// TwinCAT 3 PLC project M1L1_PLC
// ProgramVersion: 3.1.4022.7
// libraries:
//   LCLS General, * (SLAC)
//   Tc2_ControllerToolbox, * (Beckhoff Automation GmbH)
//   Tc2_MC2, * (Beckhoff Automation GmbH)
//   Tc2_SerialCom, * (Beckhoff Automation GmbH)
//   Tc2_Standard, * (Beckhoff Automation GmbH)
//   Tc2_System, * (Beckhoff Automation GmbH)
//   Tc2_Utilities, * (Beckhoff Automation GmbH)
//   Tc3_Module, * (Beckhoff Automation GmbH)
//   VisuDialogs
//   lcls-twincat-motion,0.0.0,SLAC
// project tree:
//   Common/DUTs/ E_PiezoControl.TcDUT (not stored), E_PitchControl.TcDUT (not stored), HOMS_PitchMechanism.TcDUT, ST_AbstractAxis.TcDUT (not stored), ST_HOMSStepper.TcDUT (not stored), ST_PiezoAxis.TcDUT
//   Common/POUs/Helpers/ FB_PI_E621_SerialDriver.TcPOU (not stored), FB_PI_E621_SerialTransaction.TcPOU (not stored), MC_SmoothMover.TcPOU (not stored), WithinRange.TcPOU (not stored)
//   Common/POUs/HOMS_FBs/ FB_PiezoControl.TcPOU (not stored), FB_PitchControl.TcPOU (not stored)
//   DUTs/ DUT_MotionStage_Extras.TcDUT (not stored)
//   / GlobalTextList.TcGTLO, PiezoDriver.TcTTO, PlcTask.TcTTO (not stored), Visualization Manager.TcVMO (not stored)
//   GVLs/ GVL_COM_Buffers.TcGVL (not stored), GVL_Constants.TcGVL (not stored), GVL_Devices.TcGVL, GVL_SerialIO.TcGVL (not stored)
//   POUs/ MAIN.TcPOU
//   POUs/Serial Comm/ PiezoSerial.TcPOU (not stored), P_Serial_Com.TcPOU (not stored)
//   VISUs/ Visualization.TcVIS, VISU_MotionStage.TcVIS
// real-time tasks:
//   TASK PlcTask: cycle T#10ms, priority 20, ADS port 350
//   TASK serial_com: cycle T#10ms, priority 21, ADS port 351
//   TASK PiezoDriver: cycle T#1ms, priority 3, ADS port 352
//   TASK SerialIO: cycle T#2ms, priority 1, ADS port 353
// motion (NC):
//   TASK NC-Task 1 SAF: cycle T#2ms, priority 4, ADS port 501
//   TASK NC-Task 1 SVB: cycle T#10ms, priority 8, ADS port 511
//   AXIS y_up (id 6)
//     General: UnitName=um
//     Dynamic: Acceleration=5050, Deceleration=5050, Jerk=5100500, DelayTime=0.008
//     Velo: Maximum=100
//     OtherSettings: AllowMotionCmdToSlave=true
//     encoder EncType=29
//       EncPara: ScaleFactorNumerator=1, ScaleFactorDenominator=1000, MaxCount=#xffffffff
//         SoftEndMinControl: Enable=true, Range=10000
//         SoftEndMaxControl: Enable=true, Range=79999
//         Inc: RefSoftSyncMask=#x0000ffff
//     drive DrvType=24
//       DrvPara: Inverse=true
//         Analog: VeloReferenz=500
//         TimeComp: TaskDelayCycles=1
//     controller CtrType=3
//       CtrPara: PriorControlFactor=1
//         PosDiffControl: Range=50, Time=0.2
//         PID: PosTn=0.005, PosIOutputLimit=0.0001, PosDOutputLimit=0, PosIDisableWhenMoving=true, DeadBandPosition=0.001
//         Observer: BandWidth=20
//   AXIS y_dwn (id 7)
//     General: UnitName=um
//     Dynamic: Acceleration=5050, Deceleration=5050, Jerk=5100500, DelayTime=0.008
//     Velo: Maximum=100
//     OtherSettings: AllowMotionCmdToSlave=true
//     encoder EncType=29
//       EncPara: ScaleFactorNumerator=1, ScaleFactorDenominator=1000, MaxCount=#xffffffff
//         SoftEndMinControl: Enable=true, Range=9000
//         SoftEndMaxControl: Enable=true, Range=79551
//         Inc: RefSoftSyncMask=#x0000ffff
//     drive DrvType=24
//       DrvPara: Inverse=true
//         Analog: VeloReferenz=500
//         TimeComp: TaskDelayCycles=1
//     controller CtrType=3
//       CtrPara: PriorControlFactor=1
//         PosDiffControl: Range=50, Time=0.2
//         PID: PosTn=0.005, PosIOutputLimit=0.0001, PosDOutputLimit=0, PosIDisableWhenMoving=true, DeadBandPosition=0.001
//         Observer: BandWidth=20
//   AXIS x_up (id 8)
//     General: UnitName=um
//     Dynamic: AccelerationMaximum=1000, DecelerationMaximum=1000, Acceleration=1000, Deceleration=1000, Jerk=5000, DelayTime=0.008
//     Velo: Maximum=300
//     OtherSettings: AllowMotionCmdToSlave=true
//     encoder EncType=29
//       EncPara: ScaleFactorNumerator=1, ScaleFactorDenominator=1000, MaxCount=#xffffffff
//         SoftEndMinControl: Enable=true, Range=16300
//         SoftEndMaxControl: Enable=true, Range=23200
//         Inc: RefSoftSyncMask=#x0000ffff
//     drive DrvType=24
//       DrvPara: Inverse=true
//         Analog: VeloReferenz=625
//         TimeComp: TaskDelayCycles=1
//     controller CtrType=3
//       CtrPara: PriorControlFactor=1
//         PosDiffControl: Range=50, Time=0.2
//         PID: PosTn=0.005, PosIOutputLimit=0.0001, PosDOutputLimit=0, PosIDisableWhenMoving=true, DeadBandPosition=0.001
//         Observer: BandWidth=20
//   AXIS x_dwn (id 9)
//     General: UnitName=um
//     Dynamic: AccelerationMaximum=1000, DecelerationMaximum=1000, Acceleration=1000, Deceleration=1000, Jerk=5000, DelayTime=0.008
//     Velo: Maximum=300
//     OtherSettings: AllowMotionCmdToSlave=true
//     encoder EncType=29
//       EncPara: ScaleFactorNumerator=1, ScaleFactorDenominator=1000, MaxCount=#xffffffff
//         SoftEndMinControl: Enable=true, Range=17400
//         SoftEndMaxControl: Enable=true, Range=24500
//         Inc: RefSoftSyncMask=#x0000ffff
//     drive DrvType=24
//       Analog: VeloReferenz=625
//       TimeComp: TaskDelayCycles=1
//     controller CtrType=3
//       CtrPara: PriorControlFactor=1
//         PosDiffControl: Range=50, Time=0.2
//         PID: PosTn=0.005, PosIOutputLimit=0.0001, PosDOutputLimit=0, PosIDisableWhenMoving=true, DeadBandPosition=0.001
//         Observer: BandWidth=20
//   AXIS pitch (id 10)
//     General: UnitName=urad
//     Dynamic: Acceleration=64082.2, Deceleration=64082.2, Jerk=711156, DelayTime=0.008
//     Velo: Maximum=50
//     OtherSettings: AllowMotionCmdToSlave=true
//     encoder EncType=29
//       EncPara: ScaleFactorNumerator=0.00556, MaxCount=#xffffffff
//         ActPosCorrection: Time=0.008
//         Inc: RefSoftSyncMask=#x0000ffff
//     drive DrvType=24
//       DrvPara: Inverse=true
//         Analog: VeloReferenz=7042.25
//         TimeComp: TaskDelayCycles=1
//     controller CtrType=3
//       CtrPara: PriorControlFactor=1
//         PosDiffControl: Range=15, Time=0.2
//         PID: PosKp=9, PosTn=0.0006, PosTv=1.2e-05, PosIOutputLimit=0.0005, PosDOutputLimit=0.0035, AccKa=0.001, DeadBandPosition=0.1
//         Observer: BandWidth=20
// I/O:
//   DEVICE Device 1 (EtherCAT)
//   DEVICE Device 4 (EtherCAT)
// variable links:
//   Axes/pitch <-> Device 4 (EtherCAT)/Term 4 (EK1100)/Term 10 (EL7047) - PitchCoarse
//     Drive/Inputs/In/nState1 @bit 3 <-> STM Status/Status/Error
//     Drive/Inputs/In/nState1 @bit 7 <-> STM Status/Status/Motor stall
//     Drive/Inputs/In/nState1 @bit 5 <-> STM Status/Status/Moving negative
//     Drive/Inputs/In/nState1 @bit 4 <-> STM Status/Status/Moving positive
//     Drive/Inputs/In/nState1 @bit 1 <-> STM Status/Status/Ready
//     Drive/Inputs/In/nState1 <-> STM Status/Status/Ready to enable
//     Drive/Inputs/In/nState1 @bit 6 <-> STM Status/Status/Torque reduced
//     Drive/Inputs/In/nState1 @bit 2 <-> STM Status/Status/Warning
//     Drive/Inputs/In/nState2 @bit 3 <-> STM Status/Status/Digital input 1
//     Drive/Inputs/In/nState2 @bit 4 <-> STM Status/Status/Digital input 2
//     Drive/Inputs/In/nState2 @bit 5 <-> STM Status/Status/Sync error
//     Drive/Inputs/In/nState2 @bit 7 <-> STM Status/Status/TxPDO Toggle
//     Drive/Inputs/In/nState4 @bit 1 <-> WcState/InputToggle
//     Drive/Inputs/In/nState4 <-> WcState/WcState
//     Drive/Outputs/Out/nCtrl1 <-> STM Control/Control/Enable
//     Drive/Outputs/Out/nCtrl1 @bit 2 <-> STM Control/Control/Reduce torque
//     Drive/Outputs/Out/nCtrl1 @bit 1 <-> STM Control/Control/Reset
//     Drive/Outputs/Out/nCtrl2 @bit 3 <-> STM Control/Control/Digital output 1
//     Drive/Outputs/Out/nDataOut2[0] <-> STM Velocity/Velocity
//   Axes/pitch <-> Device 4 (EtherCAT)/Term 4 (EK1100)/Term 13 (EL5042) - Pitch
//     Enc/Inputs/In/nComState @bit 1 <-> WcState/InputToggle
//     Enc/Inputs/In/nComState <-> WcState/WcState
//     Enc/Inputs/In/nDataIn1 <-> FB Inputs Channel 1/Position
//     Enc/Inputs/In/nState1 @bit 12 <-> FB Inputs Channel 1/Status/Diag
//     Enc/Inputs/In/nState1 @bit 1 <-> FB Inputs Channel 1/Status/Error
//     Enc/Inputs/In/nState1 @bit 14 <-> FB Inputs Channel 1/Status/Input cycle counter
//     Enc/Inputs/In/nState1 @bit 2 <-> FB Inputs Channel 1/Status/Ready
//     Enc/Inputs/In/nState1 @bit 13 <-> FB Inputs Channel 1/Status/TxPDO State
//     Enc/Inputs/In/nState1 <-> FB Inputs Channel 1/Status/Warning
//   Axes/x_dwn <-> Device 4 (EtherCAT)/Term 4 (EK1100)/Term 12 (EL5042) - X
//     Enc/Inputs/In/nComState @bit 1 <-> WcState/InputToggle
//     Enc/Inputs/In/nComState <-> WcState/WcState
//     Enc/Inputs/In/nDataIn1 <-> FB Inputs Channel 2/Position
//     Enc/Inputs/In/nState1 @bit 12 <-> FB Inputs Channel 2/Status/Diag
//     Enc/Inputs/In/nState1 @bit 1 <-> FB Inputs Channel 2/Status/Error
//     Enc/Inputs/In/nState1 @bit 14 <-> FB Inputs Channel 2/Status/Input cycle counter
//     Enc/Inputs/In/nState1 @bit 2 <-> FB Inputs Channel 2/Status/Ready
//     Enc/Inputs/In/nState1 @bit 13 <-> FB Inputs Channel 2/Status/TxPDO State
//     Enc/Inputs/In/nState1 <-> FB Inputs Channel 2/Status/Warning
//   Axes/x_dwn <-> Device 4 (EtherCAT)/Term 4 (EK1100)/Term 9 (EL7047) - Xdwn
//     Drive/Inputs/In/nState1 @bit 3 <-> STM Status/Status/Error
//     Drive/Inputs/In/nState1 @bit 7 <-> STM Status/Status/Motor stall
//     Drive/Inputs/In/nState1 @bit 5 <-> STM Status/Status/Moving negative
//     Drive/Inputs/In/nState1 @bit 4 <-> STM Status/Status/Moving positive
//     Drive/Inputs/In/nState1 @bit 1 <-> STM Status/Status/Ready
//     Drive/Inputs/In/nState1 <-> STM Status/Status/Ready to enable
//     Drive/Inputs/In/nState1 @bit 6 <-> STM Status/Status/Torque reduced
//     Drive/Inputs/In/nState1 @bit 2 <-> STM Status/Status/Warning
//     Drive/Inputs/In/nState2 @bit 3 <-> STM Status/Status/Digital input 1
//     Drive/Inputs/In/nState2 @bit 4 <-> STM Status/Status/Digital input 2
//     Drive/Inputs/In/nState2 @bit 5 <-> STM Status/Status/Sync error
//     Drive/Inputs/In/nState2 @bit 7 <-> STM Status/Status/TxPDO Toggle
//     Drive/Inputs/In/nState4 @bit 1 <-> WcState/InputToggle
//     Drive/Inputs/In/nState4 <-> WcState/WcState
//     Drive/Outputs/Out/nCtrl1 <-> STM Control/Control/Enable
//     Drive/Outputs/Out/nCtrl1 @bit 2 <-> STM Control/Control/Reduce torque
//     Drive/Outputs/Out/nCtrl1 @bit 1 <-> STM Control/Control/Reset
//     Drive/Outputs/Out/nCtrl2 @bit 3 <-> STM Control/Control/Digital output 1
//     Drive/Outputs/Out/nDataOut2[0] <-> STM Velocity/Velocity
//   Axes/x_up <-> Device 4 (EtherCAT)/Term 4 (EK1100)/Term 12 (EL5042) - X
//     Enc/Inputs/In/nComState @bit 1 <-> WcState/InputToggle
//     Enc/Inputs/In/nComState <-> WcState/WcState
//     Enc/Inputs/In/nDataIn1 <-> FB Inputs Channel 1/Position
//     Enc/Inputs/In/nState1 @bit 12 <-> FB Inputs Channel 1/Status/Diag
//     Enc/Inputs/In/nState1 @bit 1 <-> FB Inputs Channel 1/Status/Error
//     Enc/Inputs/In/nState1 @bit 14 <-> FB Inputs Channel 1/Status/Input cycle counter
//     Enc/Inputs/In/nState1 @bit 2 <-> FB Inputs Channel 1/Status/Ready
//     Enc/Inputs/In/nState1 @bit 13 <-> FB Inputs Channel 1/Status/TxPDO State
//     Enc/Inputs/In/nState1 <-> FB Inputs Channel 1/Status/Warning
//   Axes/x_up <-> Device 4 (EtherCAT)/Term 4 (EK1100)/Term 8 (EL7047) - Xup
//     Drive/Inputs/In/nState1 @bit 3 <-> STM Status/Status/Error
//     Drive/Inputs/In/nState1 @bit 7 <-> STM Status/Status/Motor stall
//     Drive/Inputs/In/nState1 @bit 5 <-> STM Status/Status/Moving negative
//     Drive/Inputs/In/nState1 @bit 4 <-> STM Status/Status/Moving positive
//     Drive/Inputs/In/nState1 @bit 1 <-> STM Status/Status/Ready
//     Drive/Inputs/In/nState1 <-> STM Status/Status/Ready to enable
//     Drive/Inputs/In/nState1 @bit 6 <-> STM Status/Status/Torque reduced
//     Drive/Inputs/In/nState1 @bit 2 <-> STM Status/Status/Warning
//     Drive/Inputs/In/nState2 @bit 3 <-> STM Status/Status/Digital input 1
//     Drive/Inputs/In/nState2 @bit 4 <-> STM Status/Status/Digital input 2
//     Drive/Inputs/In/nState2 @bit 5 <-> STM Status/Status/Sync error
//     Drive/Inputs/In/nState2 @bit 7 <-> STM Status/Status/TxPDO Toggle
//     Drive/Inputs/In/nState4 @bit 1 <-> WcState/InputToggle
//     Drive/Inputs/In/nState4 <-> WcState/WcState
//     Drive/Outputs/Out/nCtrl1 <-> STM Control/Control/Enable
//     Drive/Outputs/Out/nCtrl1 @bit 2 <-> STM Control/Control/Reduce torque
//     Drive/Outputs/Out/nCtrl1 @bit 1 <-> STM Control/Control/Reset
//     Drive/Outputs/Out/nCtrl2 @bit 3 <-> STM Control/Control/Digital output 1
//     Drive/Outputs/Out/nDataOut2[0] <-> STM Velocity/Velocity
//   Axes/y_dwn <-> Device 4 (EtherCAT)/Term 4 (EK1100)/Term 11 (EL5042) - Y
//     Enc/Inputs/In/nComState @bit 1 <-> WcState/InputToggle
//     Enc/Inputs/In/nComState <-> WcState/WcState
//     Enc/Inputs/In/nDataIn1 <-> FB Inputs Channel 2/Position
//     Enc/Inputs/In/nState1 @bit 12 <-> FB Inputs Channel 2/Status/Diag
//     Enc/Inputs/In/nState1 @bit 1 <-> FB Inputs Channel 2/Status/Error
//     Enc/Inputs/In/nState1 @bit 14 <-> FB Inputs Channel 2/Status/Input cycle counter
//     Enc/Inputs/In/nState1 @bit 2 <-> FB Inputs Channel 2/Status/Ready
//     Enc/Inputs/In/nState1 @bit 13 <-> FB Inputs Channel 2/Status/TxPDO State
//     Enc/Inputs/In/nState1 <-> FB Inputs Channel 2/Status/Warning
//   Axes/y_dwn <-> Device 4 (EtherCAT)/Term 4 (EK1100)/Term 7 (EL7047) - Ydwn
//     Drive/Inputs/In/nState1 @bit 3 <-> STM Status/Status/Error
//     Drive/Inputs/In/nState1 @bit 7 <-> STM Status/Status/Motor stall
//     Drive/Inputs/In/nState1 @bit 5 <-> STM Status/Status/Moving negative
//     Drive/Inputs/In/nState1 @bit 4 <-> STM Status/Status/Moving positive
//     Drive/Inputs/In/nState1 @bit 1 <-> STM Status/Status/Ready
//     Drive/Inputs/In/nState1 <-> STM Status/Status/Ready to enable
//     Drive/Inputs/In/nState1 @bit 6 <-> STM Status/Status/Torque reduced
//     Drive/Inputs/In/nState1 @bit 2 <-> STM Status/Status/Warning
//     Drive/Inputs/In/nState2 @bit 3 <-> STM Status/Status/Digital input 1
//     Drive/Inputs/In/nState2 @bit 4 <-> STM Status/Status/Digital input 2
//     Drive/Inputs/In/nState2 @bit 5 <-> STM Status/Status/Sync error
//     Drive/Inputs/In/nState2 @bit 7 <-> STM Status/Status/TxPDO Toggle
//     Drive/Inputs/In/nState4 @bit 1 <-> WcState/InputToggle
//     Drive/Inputs/In/nState4 <-> WcState/WcState
//     Drive/Outputs/Out/nCtrl1 <-> STM Control/Control/Enable
//     Drive/Outputs/Out/nCtrl1 @bit 2 <-> STM Control/Control/Reduce torque
//     Drive/Outputs/Out/nCtrl1 @bit 1 <-> STM Control/Control/Reset
//     Drive/Outputs/Out/nCtrl2 @bit 3 <-> STM Control/Control/Digital output 1
//     Drive/Outputs/Out/nDataOut2[0] <-> STM Velocity/Velocity
//   Axes/y_up <-> Device 4 (EtherCAT)/Term 4 (EK1100)/Term 11 (EL5042) - Y
//     Enc/Inputs/In/nComState @bit 1 <-> WcState/InputToggle
//     Enc/Inputs/In/nComState <-> WcState/WcState
//     Enc/Inputs/In/nDataIn1 <-> FB Inputs Channel 1/Position
//     Enc/Inputs/In/nState1 @bit 12 <-> FB Inputs Channel 1/Status/Diag
//     Enc/Inputs/In/nState1 @bit 1 <-> FB Inputs Channel 1/Status/Error
//     Enc/Inputs/In/nState1 @bit 14 <-> FB Inputs Channel 1/Status/Input cycle counter
//     Enc/Inputs/In/nState1 @bit 2 <-> FB Inputs Channel 1/Status/Ready
//     Enc/Inputs/In/nState1 @bit 13 <-> FB Inputs Channel 1/Status/TxPDO State
//     Enc/Inputs/In/nState1 <-> FB Inputs Channel 1/Status/Warning
//   Axes/y_up <-> Device 4 (EtherCAT)/Term 4 (EK1100)/Term 6 (EL7047) - Yup
//     Drive/Inputs/In/nState1 @bit 3 <-> STM Status/Status/Error
//     Drive/Inputs/In/nState1 @bit 7 <-> STM Status/Status/Motor stall
//     Drive/Inputs/In/nState1 @bit 5 <-> STM Status/Status/Moving negative
//     Drive/Inputs/In/nState1 @bit 4 <-> STM Status/Status/Moving positive
//     Drive/Inputs/In/nState1 @bit 1 <-> STM Status/Status/Ready
//     Drive/Inputs/In/nState1 <-> STM Status/Status/Ready to enable
//     Drive/Inputs/In/nState1 @bit 6 <-> STM Status/Status/Torque reduced
//     Drive/Inputs/In/nState1 @bit 2 <-> STM Status/Status/Warning
//     Drive/Inputs/In/nState2 @bit 3 <-> STM Status/Status/Digital input 1
//     Drive/Inputs/In/nState2 @bit 4 <-> STM Status/Status/Digital input 2
//     Drive/Inputs/In/nState2 @bit 5 <-> STM Status/Status/Sync error
//     Drive/Inputs/In/nState2 @bit 7 <-> STM Status/Status/TxPDO Toggle
//     Drive/Inputs/In/nState4 @bit 1 <-> WcState/InputToggle
//     Drive/Inputs/In/nState4 <-> WcState/WcState
//     Drive/Outputs/Out/nCtrl1 <-> STM Control/Control/Enable
//     Drive/Outputs/Out/nCtrl1 @bit 2 <-> STM Control/Control/Reduce torque
//     Drive/Outputs/Out/nCtrl1 @bit 1 <-> STM Control/Control/Reset
//     Drive/Outputs/Out/nCtrl2 @bit 3 <-> STM Control/Control/Digital output 1
//     Drive/Outputs/Out/nDataOut2[0] <-> STM Velocity/Velocity
//   M1L1_PLC Instance <-> Device 1 (EtherCAT)/Term 1 (EK1200)/Term 2 (EL1004)
//     PlcTask Inputs/MAIN.bSTOEnable1 <-> Channel 1/Input
//     PlcTask Inputs/MAIN.bSTOEnable2 <-> Channel 2/Input
//   M1L1_PLC Instance <-> Device 4 (EtherCAT)/Term 4 (EK1100)/Term 10 (EL7047) - PitchCoarse
//     PlcTask Inputs/GVL_Devices.M5.bLimitBackwardEnable <-> STM Status/Status/Digital input 2
//     PlcTask Inputs/GVL_Devices.M5.bLimitForwardEnable <-> STM Status/Status/Digital input 1
//   M1L1_PLC Instance <-> Device 4 (EtherCAT)/Term 4 (EK1100)/Term 11 (EL5042) - Y
//     PlcTask Inputs/MAIN.y_dwn_enc/Count <-> FB Inputs Channel 2/Position
//     PlcTask Inputs/MAIN.y_up_enc/Count <-> FB Inputs Channel 1/Position
//   M1L1_PLC Instance <-> Device 4 (EtherCAT)/Term 4 (EK1100)/Term 12 (EL5042) - X
//     PlcTask Inputs/MAIN.x_dwn_enc/Count <-> FB Inputs Channel 2/Position
//     PlcTask Inputs/MAIN.x_up_enc/Count <-> FB Inputs Channel 1/Position
//   M1L1_PLC Instance <-> Device 4 (EtherCAT)/Term 4 (EK1100)/Term 13 (EL5042) - Pitch
//     PlcTask Inputs/GVL_Devices.M1L0_Pitch.diEncCnt <-> FB Inputs Channel 1/Position
//   M1L1_PLC Instance <-> Device 4 (EtherCAT)/Term 4 (EK1100)/Term 14 (EL6001) - PitchFine
//     PlcTask Inputs/GVL_SerialIO.Serial_P1_stComIn/D[{0..21}] <-> COM Inputs/Data In {0..21}  (22 links)
//     PlcTask Inputs/GVL_SerialIO.Serial_P1_stComIn/Status <-> COM Inputs/Status
//     PlcTask Outputs/GVL_SerialIO.Serial_P1_stComOut/Ctrl <-> COM Outputs/Ctrl
//     PlcTask Outputs/GVL_SerialIO.Serial_P1_stComOut/D[{0..21}] <-> COM Outputs/Data Out {0..21}  (22 links)
//   M1L1_PLC Instance <-> Device 4 (EtherCAT)/Term 4 (EK1100)/Term 6 (EL7047) - Yup
//     PlcTask Inputs/GVL_Devices.M1.bLimitBackwardEnable <-> STM Status/Status/Digital input 2
//     PlcTask Inputs/GVL_Devices.M1.bLimitForwardEnable <-> STM Status/Status/Digital input 1
//   M1L1_PLC Instance <-> Device 4 (EtherCAT)/Term 4 (EK1100)/Term 7 (EL7047) - Ydwn
//     PlcTask Inputs/GVL_Devices.M2.bLimitBackwardEnable <-> STM Status/Status/Digital input 2
//     PlcTask Inputs/GVL_Devices.M2.bLimitForwardEnable <-> STM Status/Status/Digital input 1
//   M1L1_PLC Instance <-> Device 4 (EtherCAT)/Term 4 (EK1100)/Term 8 (EL7047) - Xup
//     PlcTask Inputs/GVL_Devices.M3.bLimitBackwardEnable <-> STM Status/Status/Digital input 2
//     PlcTask Inputs/GVL_Devices.M3.bLimitForwardEnable <-> STM Status/Status/Digital input 1
//   M1L1_PLC Instance <-> Device 4 (EtherCAT)/Term 4 (EK1100)/Term 9 (EL7047) - Xdwn
//     PlcTask Inputs/GVL_Devices.M4.bLimitBackwardEnable <-> STM Status/Status/Digital input 2
//     PlcTask Inputs/GVL_Devices.M4.bLimitForwardEnable <-> STM Status/Status/Digital input 1
//   M1L1_PLC Instance <-> NC-Task 1 SAF/Axes/pitch
//     PlcTask Inputs/GVL_Devices.M5.Axis.NcToPlc <-> Outputs/ToPlc
//     PlcTask Outputs/GVL_Devices.M5.Axis.PlcToNc <-> Inputs/FromPlc
//   M1L1_PLC Instance <-> NC-Task 1 SAF/Axes/x_dwn
//     PlcTask Inputs/GVL_Devices.M4.Axis.NcToPlc <-> Outputs/ToPlc
//     PlcTask Outputs/GVL_Devices.M4.Axis.PlcToNc <-> Inputs/FromPlc
//   M1L1_PLC Instance <-> NC-Task 1 SAF/Axes/x_up
//     PlcTask Inputs/GVL_Devices.M3.Axis.NcToPlc <-> Outputs/ToPlc
//     PlcTask Outputs/GVL_Devices.M3.Axis.PlcToNc <-> Inputs/FromPlc
//   M1L1_PLC Instance <-> NC-Task 1 SAF/Axes/y_dwn
//     PlcTask Inputs/GVL_Devices.M2.Axis.NcToPlc <-> Outputs/ToPlc
//     PlcTask Outputs/GVL_Devices.M2.Axis.PlcToNc <-> Inputs/FromPlc
//   M1L1_PLC Instance <-> NC-Task 1 SAF/Axes/y_up
//     PlcTask Inputs/GVL_Devices.M1.Axis.NcToPlc <-> Outputs/ToPlc
//     PlcTask Outputs/GVL_Devices.M1.Axis.PlcToNc <-> Inputs/FromPlc

CONFIGURATION M1L1_PLC
    RESOURCE PLC ON TwinCAT3
        TASK PiezoDriver(INTERVAL := T#1ms, PRIORITY := 3);
        PROGRAM PiezoSerial WITH PiezoDriver : PiezoSerial;
    END_RESOURCE
END_CONFIGURATION

// ---- Common/DUTs/HOMS_PitchMechanism.TcDUT
TYPE HOMS_PitchMechanism :
STRUCT
	Piezo	:	ST_PiezoAxis;	//Piezo
	Axis	:	ST_AbstractAxis; //Abstract pitch axis
//	Stepper	:	ST_HOMSStepper; //Pitch stepper axis

	(* Soft limits, egu urad *)
	ReqPosLimHi	:	REAL;
	ReqPosLimLo	:	REAL;


	(* Hard limits, egu INC *)
	(* These are discovered during installation, and represent encoder ticks, unbiased *)
	(* We changed to these when our pitch mechanism limit switches were insufficient for
	good control. They had too much hysteresis/ lack of precision. At this point the limit
	switches are ignored, and instead their function is carried out by these. *)
	diEncPosLimHi	:	LINT;
	diEncPosLimLo	:	LINT;
	//Raw encoder count
	diEncCnt	AT %I*	:	LINT;
	
	
END_STRUCT
END_TYPE

// ---- Common/DUTs/ST_PiezoAxis.TcDUT
TYPE ST_PiezoAxis :
STRUCT
	(* IO *)
		//Readback
		sIdn				:	STRING; //Identity
		iCurError			:	INT; //Current error code, should be 0 most of the time
		iLastError			:	INT; //Last error code, for history
		rActVoltage			:	REAL; //Actual voltage
		rLastReqVoltage		:	REAL; //Last requested piezo voltage
		//Control
		rSetVoltage			:	REAL; //this parameter is set by the control loop/ voltage mode
		sAxis				:   STRING :='A'; //Axis, e.g. A, B, C...A if single unit	
		//Summaries
		xTimeout	:	BOOL;
		xDriverError		:	BOOL; //Summary of any driver errors
	
	(* Operation *)
		xEnable	:	BOOL; //Enable control.
		(* Note: Voltage mode and Idle mode overrides "DirectPiezoMode" of FB_PitchControl *)
		xVoltageMode	:	BOOL; //Voltage mode gives direct access to piezo voltage, false means closed loop position acquisition (see FB_PitchControl for piezo and stepper separation)
		xIdleMode	:	BOOL; //Use to put the piezo at half-stroke
		rReqVoltage : REAL; //Requested piezo voltage in voltage mode
		rReqAbsPos	:	LREAL; //Requested Position, latched at rising StartAbsMov
		xStop	:	BOOL;	//Stops piezo and holds position
	
	
	(* Control Parameters *)
		rActPos	:	LREAL; //Encoder Readback
		//Pitch piezo dmove range (urad)
		rPiezoDmovRange		:	REAL := 1;
		stPIParams	:	ST_CTRL_PI_PARAMS := (
			tCtrlCycleTime := T#0MS, 
			tTaskCycleTime := T#0MS, 
			tTn       := T#1S, 
			fKp      := 0.25, 
			fOutMaxLimit := 1, 
			fOutMinLimit := -1, 
			bARWOnIPartOnly := FALSE);
	
	(* Voltage ranges, come from specifications of the driver *)
		UpperVoltage	:	REAL := cPiezoMaxVoltage; // E-816 has no software limits
		LowerVoltage	:	REAL := cPiezoMinVoltage; // E-816 has no software limits
END_STRUCT
END_TYPE

// ---- GVLs/GVL_Devices.TcGVL
VAR_GLOBAL
	// Axes
    M1: DUT_MotionStage:=(nCommand:=3); // Yup
	M2: DUT_MotionStage:=(nCommand:=3); // Ydwn
	M3: DUT_MotionStage:=(nCommand:=3); // Xup
	M4: DUT_MotionStage:=(nCommand:=3); // Xdwn
	M5: DUT_MotionStage:=(nCommand:=3); // PitchCoarse
	M1_Extras : DUT_MotionStage_Extras;
	M2_Extras : DUT_MotionStage_Extras;
	M3_Extras : DUT_MotionStage_Extras;
	M4_Extras : DUT_MotionStage_Extras;
	M5_Extras : DUT_MotionStage_Extras;

	M1L0_Pitch	    :	HOMS_PitchMechanism := (
		ReqPosLimHi := 56000,
		ReqPosLimLo := 54150,
		diEncPosLimHi := 10126850,
		diEncPosLimLo := 9727550);
END_VAR

// ---- POUs/MAIN.TcPOU
PROGRAM MAIN
VAR
(*
    M1: DUT_MotionStage:=(nCommand:=3); // Yup
	M2: DUT_MotionStage:=(nCommand:=3); // Ydwn
	M3: DUT_MotionStage:=(nCommand:=3); // Xup
	M4: DUT_MotionStage:=(nCommand:=3); // Xdwn
	M5: DUT_MotionStage:=(nCommand:=3); // PitchCoarse
*)
	
	fbMotionStage_x_up, fbMotionStage_x_dwn, fbMotionStage_y_up, fbMotionStage_y_dwn, fbMotionStage_pitch : FB_MotionStage;

	bSTOEnable1 AT %I* : BOOL;
	bSTOEnable2 AT %I* : BOOL;
	x_up_enc  AT %I*: ST_RenishawAbsEnc;
	x_dwn_enc  AT %I*: ST_RenishawAbsEnc;
	y_up_enc  AT %I*: ST_RenishawAbsEnc;
	y_dwn_enc  AT %I*: ST_RenishawAbsEnc;

	// Auto coupling function block
	fbAutoCoupleX : FB_GantryAutoCoupling;
	fbAutoCoupleY : FB_GantryAutoCoupling;
	bExecuteCoupleX : BOOL;
	bExecuteCoupleY : BOOL;
	bExecuteDecoupleX : BOOL;
	bExecuteDecoupleY : BOOL;
	bGantryAlreadyCoupledX : BOOL;
	bGantryAlreadyCoupledY : BOOL;
	
	// Gantry variables
	nCurrGantryX : LINT;
	nCurrGantryY : LINT;
	nGantryTolX : LINT := 75000;
	nGantryTolY : LINT := 75000;
	fCurrGantryX_um : LREAL;
	fCurrGantryY_um : LREAL;
	
	// Piezo Control:
	fbPitchControl : FB_PitchControl;

	// Expert mode permits direct access to individual acutators.
	ExpertMode	:	BOOL := FALSE;
	PitchManualMode: BOOL := FALSE;
END_VAR

// M1K3
// Buttons to enable motors: write 0 to enable, 2 to disable
M1.nEnableMode; // Yup
M2.nEnableMode; // Ydwn
M3.nEnableMode; // Xup
M4.nEnableMode; // Xdwn
M5.nEnableMode; // PitchCoarse

// M1K3 Ref Vals
y_up_enc.Ref := 108743550;
y_dwn_enc.Ref := 108243370;
x_up_enc.Ref := 19628100;
x_dwn_enc.Ref := 20865800;

// Gantry Differences to monitor
nCurrGantryY := ((ULINT_TO_LINT(y_up_enc.Count) - ULINT_TO_LINT(y_up_enc.Ref)) - (ULINT_TO_LINT(y_dwn_enc.Count) - ULINT_TO_LINT(y_dwn_enc.Ref)));
fCurrGantryY_um := LINT_TO_LREAL(nCurrGantryY)/1000.0;
nCurrGantryX := ((ULINT_TO_LINT(x_up_enc.Count) - ULINT_TO_LINT(x_up_enc.Ref)) - (ULINT_TO_LINT(x_dwn_enc.Count) - ULINT_TO_LINT(x_dwn_enc.Ref)));
fCurrGantryX_um := LINT_TO_LREAL(nCurrGantryX)/1000.0;

// E-stop
M1.bHardwareEnable := bSTOEnable1 AND bSTOEnable2;
M2.bHardwareEnable := bSTOEnable1 AND bSTOEnable2;
M3.bHardwareEnable := bSTOEnable1 AND bSTOEnable2;
M4.bHardwareEnable := bSTOEnable1 AND bSTOEnable2;
M5.bHardwareEnable := bSTOEnable1 AND bSTOEnable2;


// Start Autocoupling
fbAutoCoupleX(nGantryTol:=nGantryTolX, Master:=M3, MasterEnc:=x_up_enc, Slave:=M4,
	          SlaveEnc:=x_dwn_enc, bExecuteCouple:=bExecuteCoupleX,
              bExecuteDecouple:=bExecuteDecoupleX,
              bGantryAlreadyCoupled=>bGantryAlreadyCoupledX);

fbAutoCoupleY(nGantryTol:=nGantryTolY, Master:=M1, MasterEnc:=y_up_enc, Slave:=M2,
	          SlaveEnc:=y_dwn_enc, bExecuteCouple:=bExecuteCoupleY,
              bExecuteDecouple:=bExecuteDecoupleY,
			  bGantryAlreadyCoupled=>bGantryAlreadyCoupledY);

fbMotionStage_y_up  (stMotionStage:=M1);
fbMotionStage_y_dwn (stMotionStage:=M2);
fbMotionStage_x_up  (stMotionStage:=M3);
fbMotionStage_x_dwn (stMotionStage:=M4);
fbMotionStage_pitch (stMotionStage:=M5);

// Pitch Control
//fbPitchControl(Pitch:=M1L0_Pitch,
//                   DirectPiezoMode:=(ExpertMode AND PitchManualMode),
//                   q_xDone=>M1L0_Pitch.Axis.bDone,
//                   q_xBusy=>M1L0_Pitch.Axis.bBusy);

END_PROGRAM

// ---- GlobalTextList.TcGTLO
TEXTLIST GlobalTextList
  234 = '%f'
  608 = '%X'
  600 = '+'
  594 = '-'
  604 = '0 = Default Acceleration'
  606 = '0 = Default Deceleration'
  603 = 'Acceleration: %f'
  963 = 'Already Coupled: %f'
  598 = 'Clear'
  592 = 'Control'
  322 = 'Couple Motors'
  336 = 'Couple Status: 0 = Decoupled, 1 = Coupled'
  964 = 'Couple Status: TRUE if coupled'
  678 = 'Current Gantry Difference (Axilon): %f'
  321 = 'Current Gantry Difference in um'
  320 = 'Current Gantry Difference: %f'
  235 = 'Current Position'
  605 = 'Deceleration: %f'
  331 = 'Decouple Motors'
  333 = 'Disable'
  334 = 'Enable'
  329 = 'Enable Mode: %f'
  335 = 'Enable Status: 0 = Enabled, 2 = Disabled'
  337 = 'Ensure motors are coupled before attempting motion!'
  609 = 'Error Code'
  607 = 'Error:'
  596 = 'GO'
  597 = 'GO to set position'
  236 = 'High Limit Hit Indicator'
  233 = 'Low Limit Hit Indicator'
  591 = 'Moving:'
  326 = 'Pitch - MASTER'
  323 = 'Press To Couple Motors'
  332 = 'Press To Decouple Motors for independent control'
  593 = 'Set Position'
  601 = 'Settings'
  232 = 'Status'
  595 = 'Step Size'
  599 = 'STOP'
  327 = 'Units: um'
  328 = 'Units: urad'
  602 = 'Velocity: %f'
  330 = 'Write 0 to Enable, 2 to Disable'
  325 = 'Xdwn - SLAVE'
  324 = 'Xup - MASTER'
  734 = 'Ydwn - SLAVE'
  961 = 'Yleft - MASTER'
  962 = 'Yright - SLAVE'
  861 = 'Yup - MASTER'
END_TEXTLIST

// ---- VISUs/Visualization.TcVIS
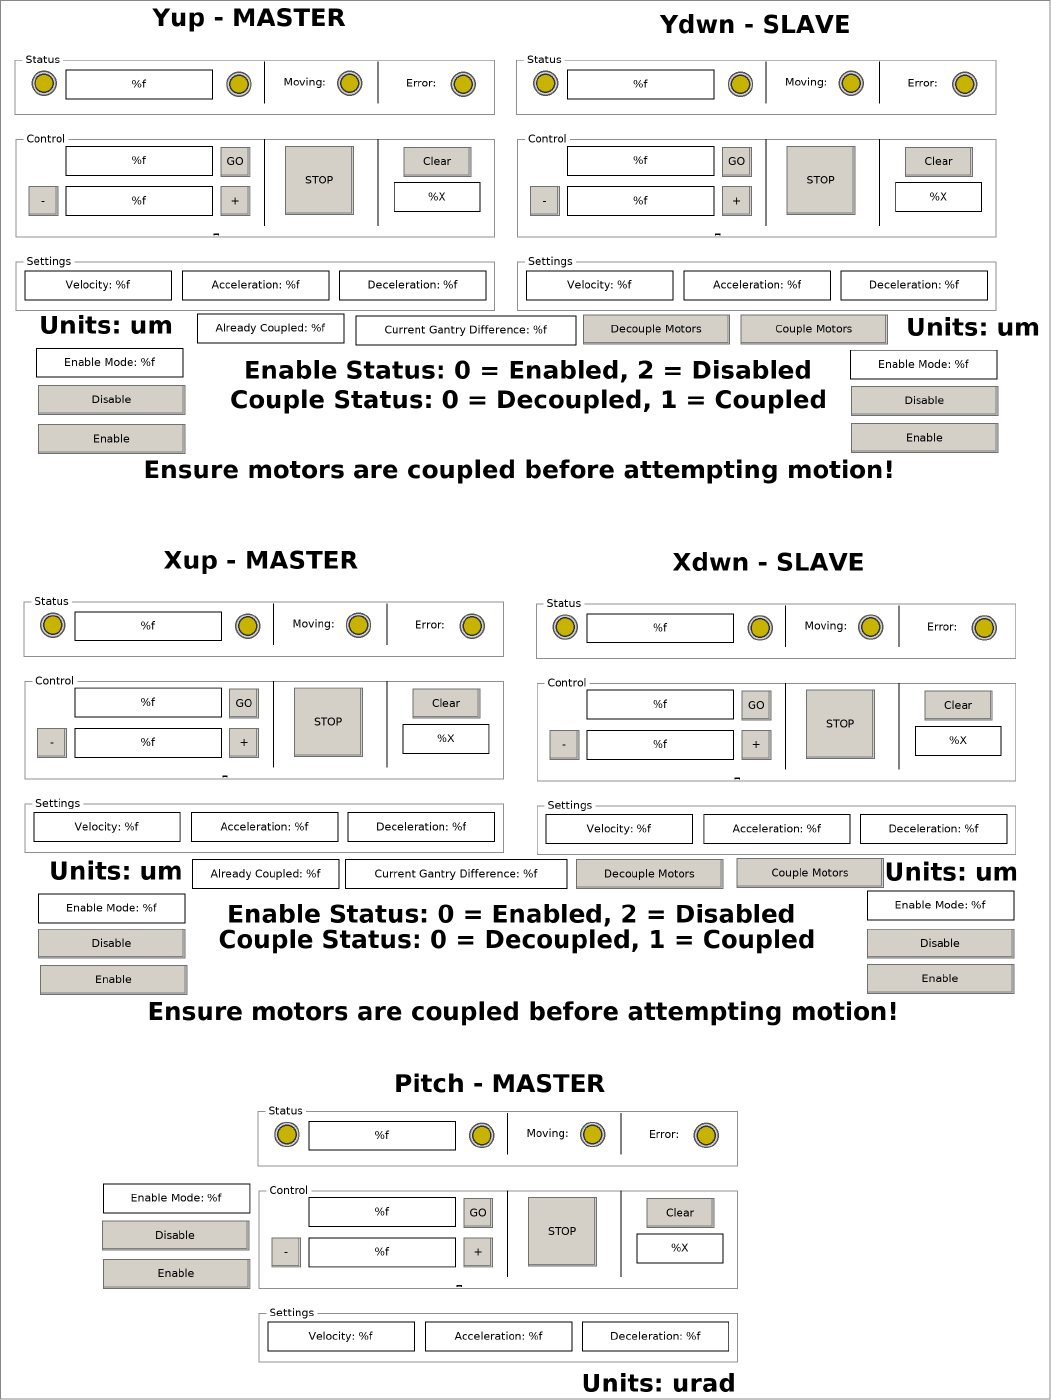
VISUALIZATION Visualization  // 1073x1429
    Label (14,2 481x31), "Yup - MASTER"
    Frame (0,36 520x300)
        shows VISU_MotionStage(VisuMotionStage := MAIN.M1, Extras := MAIN.M1_Extras)
    Frame (512,36 520x300)
        shows VISU_MotionStage(VisuMotionStage := MAIN.M2, Extras := MAIN.M2_Extras)
    Label (531,9 481x31), "Ydwn - SLAVE"
    Rectangle (201,320 150x30), "Already Coupled: %f", tooltip "Couple Status: TRUE if coupled", text variable: MAIN.bGantryAlreadyCoupledY
    Rectangle (363,322 225x30), "Current Gantry Difference: %f", tooltip "Current Gantry Difference in um", text variable: MAIN.fCurrGantryY_um
    Button (756,321 150x30), "Couple Motors", tooltip "Press To Couple Motors", text variable: MAIN.bExecuteCoupleY
        OnMouseDown: execute { MAIN.bExecuteCoupleY := TRUE; }
    Frame (9,589 520x300)
        shows VISU_MotionStage(VisuMotionStage := MAIN.M3, Extras := MAIN.M3_Extras)
    Label (26,556 481x31), "Xup - MASTER"
    Frame (532,591 520x300)
        shows VISU_MotionStage(VisuMotionStage := MAIN.M4, Extras := MAIN.M4_Extras)
    Label (544,558 481x31), "Xdwn - SLAVE"
    Rectangle (196,877 150x30), "Already Coupled: %f", tooltip "Couple Status: TRUE if coupled", text variable: MAIN.bGantryAlreadyCoupledX
    Rectangle (352,877 227x30), "Current Gantry Difference: %f", tooltip "Current Gantry Difference in um", text variable: MAIN.fCurrGantryX_um
    Frame (248,1109 520x300)
        shows VISU_MotionStage(VisuMotionStage := MAIN.M5, Extras := MAIN.M5_Extras)
    Label (270,1090 481x31), "Pitch - MASTER"
    Label (31,316 155x31), "Units: um"
    Label (916,318 155x31), "Units: um"
    Label (41,873 155x31), "Units: um"
    Label (894,874 155x31), "Units: um"
    Label (595,1396 155x31), "Units: urad"
    Rectangle (37,355 150x30), "Enable Mode: %f", tooltip "Write 0 to Enable, 2 to Disable", text variable: MAIN.M1.nEnableMode
    Rectangle (868,357 150x30), "Enable Mode: %f", tooltip "Write 0 to Enable, 2 to Disable", text variable: MAIN.M2.nEnableMode
    Button (595,321 150x30), "Decouple Motors", tooltip "Press To Decouple Motors for independent control"
        OnMouseDown: execute { MAIN.bExecuteDecoupleY := TRUE; }
    Button (39,393 150x30), "Disable"
        OnMouseDown: execute { MAIN.M1.nEnableMode := 2; }
    Button (39,433 150x30), "Enable", colour toggle: MAIN.bExecuteDecoupleY
        OnMouseDown: execute { MAIN.M1.nEnableMode := 0; }
    Button (869,394 150x30), "Disable"
        OnMouseDown: execute { MAIN.M2.nEnableMode := 2; }
    Button (869,432 150x30), "Enable", colour toggle: MAIN.bExecuteDecoupleY
        OnMouseDown: execute { MAIN.M2.nEnableMode := 0; }
    Button (588,877 150x30), "Decouple Motors", tooltip "Press To Decouple Motors for independent control"
        OnMouseDown: execute { MAIN.bExecuteDecoupleX := TRUE; }
    Button (752,876 150x30), "Couple Motors", tooltip "Press To Couple Motors", text variable: MAIN.bExecuteCoupleY
        OnMouseDown: execute { MAIN.bExecuteCoupleX := TRUE; }
    Rectangle (39,912 150x30), "Enable Mode: %f", tooltip "Write 0 to Enable, 2 to Disable", text variable: MAIN.M3.nEnableMode
    Button (39,948 150x30), "Disable"
        OnMouseDown: execute { MAIN.M3.nEnableMode := 2; }
    Button (41,985 150x30), "Enable", colour toggle: MAIN.bExecuteDecoupleY
        OnMouseDown: execute { MAIN.M3.nEnableMode := 0; }
    Rectangle (885,909 150x30), "Enable Mode: %f", tooltip "Write 0 to Enable, 2 to Disable", text variable: MAIN.M4.nEnableMode
    Button (885,948 150x30), "Disable"
        OnMouseDown: execute { MAIN.M4.nEnableMode := 2; }
    Button (885,984 150x30), "Enable", colour toggle: MAIN.bExecuteDecoupleY
        OnMouseDown: execute { MAIN.M4.nEnableMode := 0; }
    Rectangle (105,1208 150x30), "Enable Mode: %f", tooltip "Write 0 to Enable, 2 to Disable", text variable: MAIN.M5.nEnableMode
    Button (104,1246 150x30), "Disable"
        OnMouseDown: execute { MAIN.M5.nEnableMode := 2; }
    Button (105,1285 150x30), "Enable", colour toggle: MAIN.bExecuteDecoupleY
        OnMouseDown: execute { MAIN.M5.nEnableMode := 0; }
    Label (255,362 568x31), "Enable Status: 0 = Enabled, 2 = Disabled"
    Label (247,392 586x31), "Couple Status: 0 = Decoupled, 1 = Coupled"
    Label (238,917 568x31), "Enable Status: 0 = Enabled, 2 = Disabled"
    Label (235,943 586x31), "Couple Status: 0 = Decoupled, 1 = Coupled"
    Label (150,464 760x30), "Ensure motors are coupled before attempting motion!"
    Label (154,1017 760x30), "Ensure motors are coupled before attempting motion!"
END_VISUALIZATION

// ---- VISUs/VISU_MotionStage.TcVIS
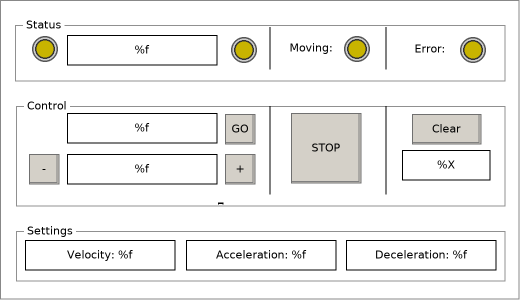
VISUALIZATION VISU_MotionStage  // 520x300
VAR_IN_OUT
	VisuMotionStage: DUT_MotionStage;
	Extras: DUT_MotionStage_Extras;
END_VAR
    GroupBox (15,17 490x64), "Status"
        Lamp1 (15,17 30x30), tooltip "Low Limit Hit Indicator", variable: Extras.bVisuLowLim, style: Lamp-Lamp1-Yellow
        Rectangle (52,18 150x30), "%f", tooltip "Current Position", text variable: VisuMotionStage.stAxisStatus.fActPosition
        Lamp1 (214,18 30x30), tooltip "High Limit Hit Indicator", variable: Extras.bVisuHighLim, style: Lamp-Lamp1-Yellow
        Lamp1 (327,17 30x30), variable: VisuMotionStage.bBusy, style: Lamp-Lamp1-Yellow
        Label (262,16 68x30), "Moving:"
        Line (371,52) (371,10)
        Lamp1 (443,18 30x30), variable: VisuMotionStage.bError, style: Lamp-Lamp1-Yellow
    Rectangle (218,203 5x0)
    GroupBox (16,98 489x108), "Control"
        Rectangle (51,15 150x30), "%f", tooltip "Set Position", text variable: VisuMotionStage.fPosition
            OnMouseDown: write the text variable via Default
        Button (13,56 30x30), "-"
            OnMouseDown: execute {
                VisuMotionStage.nCommand := 3;
                VisuMotionStage.fPosition := VisuMotionStage.stAxisStatus.fActPosition - Extras.fVisuStep;
                VisuMotionStage.bExecute := TRUE;
            }
        Rectangle (51,56 150x30), "%f", tooltip "Step Size", text variable: Extras.fVisuStep
            OnMouseDown: write the text variable via Default
        Button (209,16 30x30), "GO", tooltip "GO to set position"
            OnMouseDown: execute { VisuMotionStage.nCommand := 3; VisuMotionStage.bExecute := TRUE; }
        Line (254,96) (254,8)
        Line (370,96) (370,8)
        Button (396,16 69x30), "Clear"
            tap VisuMotionStage.bReset
        Button (275,15 70x70), "STOP", tooltip "GO to set position"
            OnMouseDown: execute { VisuMotionStage.bExecute := FALSE; }
        Button (209,56 30x30), "+"
            OnMouseDown: execute {
                VisuMotionStage.nCommand := 3;
                VisuMotionStage.fPosition := VisuMotionStage.stAxisStatus.fActPosition + Extras.fVisuStep;
                VisuMotionStage.bExecute := TRUE;
            }
    GroupBox (16,223 489x58), "Settings"
        Rectangle (9,17 150x30), "Velocity: %f", text variable: VisuMotionStage.fVelocity
            OnMouseDown: write the text variable via Default
        Rectangle (170,17 150x30), "Acceleration: %f", tooltip "0 = Default Acceleration", text variable: VisuMotionStage.fAcceleration
            OnMouseDown: write the text variable via Default
        Rectangle (330,17 150x30), "Deceleration: %f", tooltip "0 = Default Deceleration", text variable: VisuMotionStage.fDeceleration
            OnMouseDown: write the text variable via Default
    Line (270,69) (270,27)
    Label (396,34 68x30), "Error:"
    Rectangle (402,150 88x30), "%X", tooltip "Error Code", text variable: VisuMotionStage.stAxisStatus.nErrorId
END_VISUALIZATION
